PROGRAM PRG_01_PLCTASK
VAR
END_VAR

PRG_AL1L1_L2SI();
PRG_IM2L1_PPM();
PRG_SL3L1_SCATTER();
PRG_TXI_PM();

END_PROGRAM

(* stored: Version 1.1.0.1, ProductVersion 3.1.4024.6
   POU PRG_01_PLCTASK: Id {c49bac57-9deb-43fc-afb7-c59d4de2967e}, SpecialFunc None *)
